PROGRAM prgComEffIO
VAR
	fbCom		: FB_MqttCommunicator_v3;

END_VAR

fbCom(
	bConnect:= TRUE, 
	strAuthkey := 'DEV01673741737',
	sUserName:= '7faaada5-01ee-4fc7-a233-b39b42735014' , 		
	sUserPassword:= '1e6648ed-405b-46dc-9b54-28dc91eff195',
	eSavePositionCertificate:= eSavePositionOnPLC.ePostionC, 
	bConnected=> , 
	bError=> , 
	hrErrorCode=> , 
	eConnectionState=> , 
	eErrorMessage_Out=> );

END_PROGRAM

(* stored: Version 1.1.0.1, ProductVersion 3.1.4024.12
   POU prgComEffIO: Id {983c1e99-1a61-46be-bc18-1c52dda91fd9}, SpecialFunc None *)
